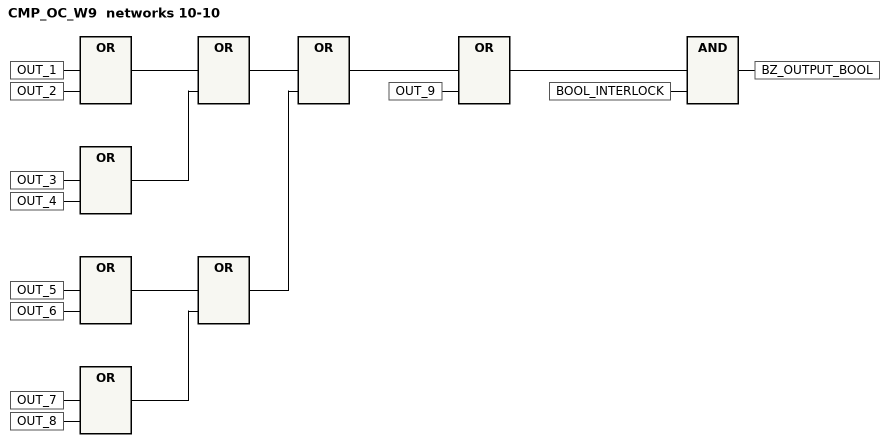
[picture p24: CMP_OC_W9 (FBD) networks 10-10]
_FBD_ (* Function Block Diagram *)
NETWORK 1
	OR(LT(WORD_1, 0), GT(WORD_1, 0)) => OUT_1
NETWORK 2
	OR(LT(WORD_2, 0), GT(WORD_2, 0)) => OUT_2
NETWORK 3
	OR(LT(WORD_3, 0), GT(WORD_3, 0)) => OUT_3
NETWORK 4
	OR(LT(WORD_4, 0), GT(WORD_4, 0)) => OUT_4
NETWORK 5
	OR(LT(WORD_5, 0), GT(WORD_5, 0)) => OUT_5
NETWORK 6
	OR(LT(WORD_6, 0), GT(WORD_6, 0)) => OUT_6
NETWORK 7
	OR(LT(WORD_7, 0), GT(WORD_7, 0)) => OUT_7
NETWORK 8
	OR(LT(WORD_8, 0), GT(WORD_8, 0)) => OUT_8
NETWORK 9
	OR(LT(WORD_9, 0), GT(WORD_9, 0)) => OUT_9
NETWORK 10
	AND(OR(OR(OR(OR(OUT_1, OUT_2), OR(OUT_3, OUT_4)), OR(OR(OUT_5, OUT_6), OR(OUT_7, OUT_8))), OUT_9), BOOL_INTERLOCK) => BZ_OUTPUT_BOOL
_END_FBD_
(* the same logic as Structured Text *)
(* Network 1 *)
OUT_1 := (WORD_1 < 0) OR (WORD_1 > 0);
(* Network 2 *)
OUT_2 := (WORD_2 < 0) OR (WORD_2 > 0);
(* Network 3 *)
OUT_3 := (WORD_3 < 0) OR (WORD_3 > 0);
(* Network 4 *)
OUT_4 := (WORD_4 < 0) OR (WORD_4 > 0);
(* Network 5 *)
OUT_5 := (WORD_5 < 0) OR (WORD_5 > 0);
(* Network 6 *)
OUT_6 := (WORD_6 < 0) OR (WORD_6 > 0);
(* Network 7 *)
OUT_7 := (WORD_7 < 0) OR (WORD_7 > 0);
(* Network 8 *)
OUT_8 := (WORD_8 < 0) OR (WORD_8 > 0);
(* Network 9 *)
OUT_9 := (WORD_9 < 0) OR (WORD_9 > 0);
(* Network 10 *)
BZ_OUTPUT_BOOL := ((((OUT_1 OR OUT_2) OR (OUT_3 OR OUT_4)) OR ((OUT_5 OR OUT_6) OR (OUT_7 OR OUT_8))) OR OUT_9) AND BOOL_INTERLOCK;
END_FUNCTION_BLOCK

(* POU DOWN_COUNT_TIMER, LD *)
FUNCTIONBLOCK DOWN_COUNT_TIMER
VAR_INPUT
	BOOL_SIGNAL_IN: BOOL;
	BOOL_TIMER_RST: BOOL;
	INT_AUTO_RST: INT;
	INT_SV_SEC: INT;
END_VAR
VAR_OUTPUT
	SIGNAL_BOOL: BOOL;
	PV_SEC_INT: INT;
END_VAR
VAR
	DF_1: R_TRIG;
	DF_2: R_TRIG;
	M1: BOOL;
	M2: BOOL;

	T100: TON;
	T101: TON;
	M100: BOOL;
	M101: BOOL;
	M200: BOOL;

	M110: BOOL;
	M300: BOOL;
END_VAR
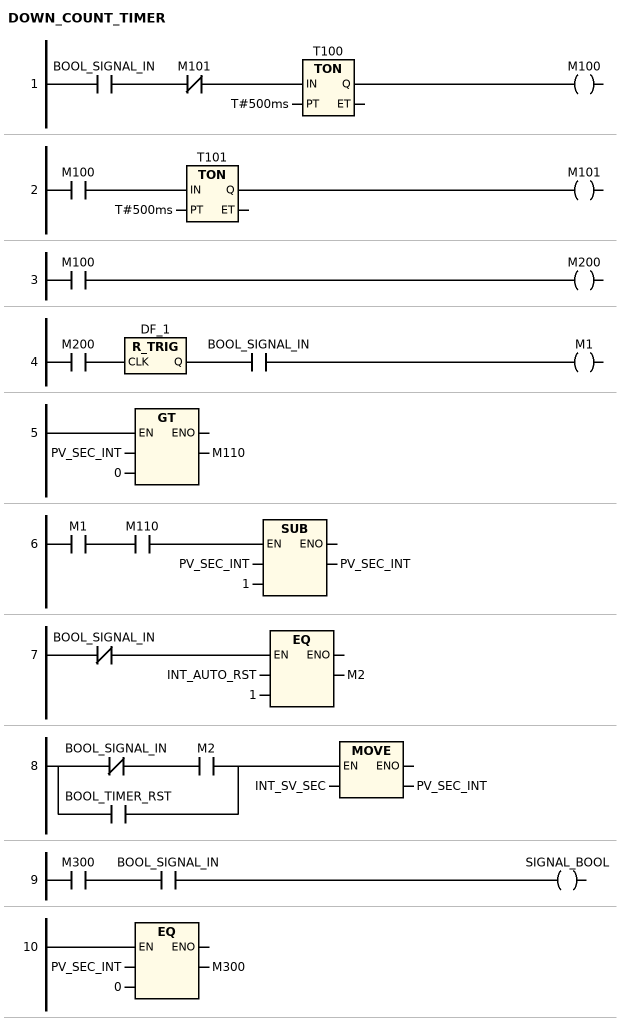
_LD_ (* Ladder Diagram *)
NETWORK 1
	[BOOL_SIGNAL_IN] - [/M101] - T100:TON(IN: *, PT: T#500ms) --- (M100)
NETWORK 2
	[M100] - T101:TON(IN: *, PT: T#500ms) --- (M101)
NETWORK 3
	[M100] --- (M200)
NETWORK 4
	[M200] - DF_1:R_TRIG(CLK: *) - [BOOL_SIGNAL_IN] --- (M1)
NETWORK 5
	*
		EN --- GT(PV_SEC_INT, 0) => M110
NETWORK 6
	[M1] - [M110]
		EN --- SUB(PV_SEC_INT, 1) => PV_SEC_INT
NETWORK 7
	[/BOOL_SIGNAL_IN]
		EN --- EQ(INT_AUTO_RST, 1) => M2
NETWORK 8
	{ [/BOOL_SIGNAL_IN] - [M2] | [BOOL_TIMER_RST] }
		EN --- MOVE(INT_SV_SEC) => PV_SEC_INT
NETWORK 9
	[M300] - [BOOL_SIGNAL_IN] --- (SIGNAL_BOOL)
NETWORK 10
	*
		EN --- EQ(PV_SEC_INT, 0) => M300
_END_LD_
(* the same logic as Structured Text *)
(* Network 1 *)
T100(IN := BOOL_SIGNAL_IN AND NOT M101, PT := T#500ms);
M100 := T100.Q;
(* Network 2 *)
T101(IN := M100, PT := T#500ms);
M101 := T101.Q;
(* Network 3 *)
M200 := M100;
(* Network 4 *)
DF_1(CLK := M200);
M1 := DF_1.Q AND BOOL_SIGNAL_IN;
(* Network 5 *)
M110 := PV_SEC_INT > 0;
(* Network 6 *)
IF M1 AND M110 THEN
	PV_SEC_INT := PV_SEC_INT - 1;
END_IF;
(* Network 7 *)
IF NOT BOOL_SIGNAL_IN THEN
	M2 := INT_AUTO_RST = 1;
END_IF;
(* Network 8 *)
IF NOT BOOL_SIGNAL_IN AND M2 OR BOOL_TIMER_RST THEN
	PV_SEC_INT := INT_SV_SEC;
END_IF;
(* Network 9 *)
SIGNAL_BOOL := M300 AND BOOL_SIGNAL_IN;
(* Network 10 *)
M300 := PV_SEC_INT = 0;
END_FUNCTION_BLOCK

(* POU CLOCK_PLS, LD *)
FUNCTION_BLOCK CLOCK_PLS
VAR_INPUT
	INT_TIME_ms : INT;

END_VAR
VAR_OUTPUT
	CLOCK_PLS_BOOL: BOOL;
END_VAR
VAR
	T0: TON;
	T1: TON;
	M0: BOOL;
	M1: BOOL;
	D0: TIME;
	D1: TIME;
END_VAR
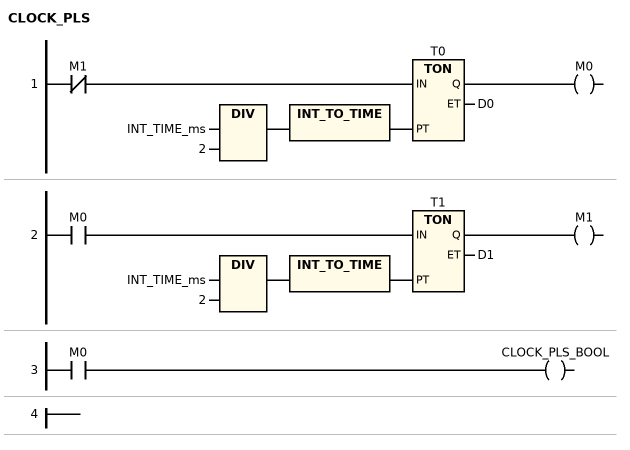
_LD_ (* Ladder Diagram *)
NETWORK 1
	[/M1] - T0:TON(IN: *, PT: INT_TO_TIME(DIV(INT_TIME_ms, 2)), ET => D0) --- (M0)
NETWORK 2
	[M0] - T1:TON(IN: *, PT: INT_TO_TIME(DIV(INT_TIME_ms, 2)), ET => D1) --- (M1)
NETWORK 3
	[M0] --- (CLOCK_PLS_BOOL)
NETWORK 4
	*
_END_LD_
(* the same logic as Structured Text *)
(* Network 1 *)
T0(IN := NOT M1, PT := INT_TO_TIME(INT_TIME_ms / 2));
D0 := T0.ET;
M0 := T0.Q;
(* Network 2 *)
T1(IN := M0, PT := INT_TO_TIME(INT_TIME_ms / 2));
D1 := T1.ET;
M1 := T1.Q;
(* Network 3 *)
CLOCK_PLS_BOOL := M0;
(* Network 4 *)
END_FUNCTION_BLOCK

(* POU DC_PID_FB, LD *)
FUNCTION_BLOCK DC_PID_FB
VAR_INPUT
	BOOL_LOW_FLOW_EN : BOOL;
	INT_HIGH_FLOW_LPM : INT;
	INT_LOW_FLOW_LPM : INT;
	INT_H_L_FLOW_RATIO : INT;
	INT_D1_LPM : INT;
	INT_D2_LPM : INT;
	INT_D3_LPM : INT;
	INT_D4_RAW : INT;
	INT_D5_RAW : INT;
	INT_D6_RAW : INT;
	INT_D1_RATIO : INT;
	INT_D2_RATIO : INT;
	INT_D3_RATIO : INT;
	INT_D4_RATIO : INT;
	INT_D5_RATIO : INT;
	INT_D6_RATIO : INT;

END_VAR

VAR_OUTPUT

	PID_FLOW_RAW : INT;
	D1_RAW_INT : INT;
	D2_RAW_INT : INT;
	D3_RAW_INT : INT;
	D4_LPM_INT : INT;
	D5_LPM_INT : INT;
	D6_LPM_INT : INT;

END_VAR
VAR
	D5EN: BOOL;
	D4EN: BOOL;
	D6EN: BOOL;
	D4REN: BOOL;
	D5REN: BOOL;
	D6REN: BOOL;
END_VAR
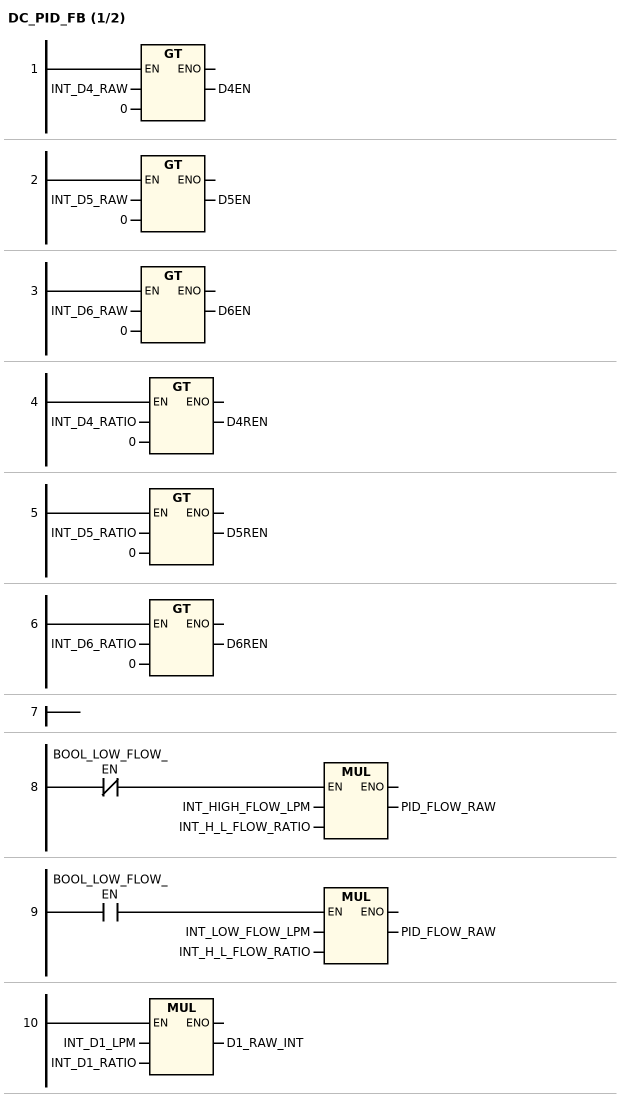
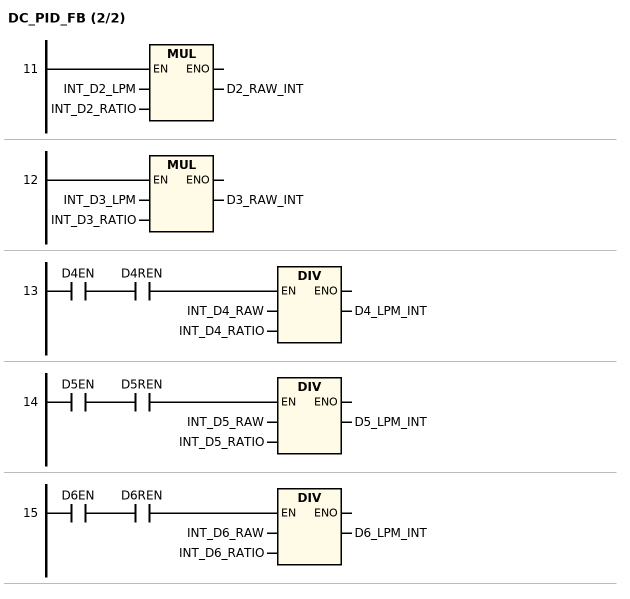
_LD_ (* Ladder Diagram *)
NETWORK 1
	*
		EN --- GT(INT_D4_RAW, 0) => D4EN
NETWORK 2
	*
		EN --- GT(INT_D5_RAW, 0) => D5EN
NETWORK 3
	*
		EN --- GT(INT_D6_RAW, 0) => D6EN
NETWORK 4
	*
		EN --- GT(INT_D4_RATIO, 0) => D4REN
NETWORK 5
	*
		EN --- GT(INT_D5_RATIO, 0) => D5REN
NETWORK 6
	*
		EN --- GT(INT_D6_RATIO, 0) => D6REN
NETWORK 7
	*
NETWORK 8
	[/BOOL_LOW_FLOW_EN]
		EN --- MUL(INT_HIGH_FLOW_LPM, INT_H_L_FLOW_RATIO) => PID_FLOW_RAW
NETWORK 9
	[BOOL_LOW_FLOW_EN]
		EN --- MUL(INT_LOW_FLOW_LPM, INT_H_L_FLOW_RATIO) => PID_FLOW_RAW
NETWORK 10
	*
		EN --- MUL(INT_D1_LPM, INT_D1_RATIO) => D1_RAW_INT
NETWORK 11
	*
		EN --- MUL(INT_D2_LPM, INT_D2_RATIO) => D2_RAW_INT
NETWORK 12
	*
		EN --- MUL(INT_D3_LPM, INT_D3_RATIO) => D3_RAW_INT
NETWORK 13
	[D4EN] - [D4REN]
		EN --- DIV(INT_D4_RAW, INT_D4_RATIO) => D4_LPM_INT
NETWORK 14
	[D5EN] - [D5REN]
		EN --- DIV(INT_D5_RAW, INT_D5_RATIO) => D5_LPM_INT
NETWORK 15
	[D6EN] - [D6REN]
		EN --- DIV(INT_D6_RAW, INT_D6_RATIO) => D6_LPM_INT
_END_LD_
(* the same logic as Structured Text *)
(* Network 1 *)
D4EN := INT_D4_RAW > 0;
(* Network 2 *)
D5EN := INT_D5_RAW > 0;
(* Network 3 *)
D6EN := INT_D6_RAW > 0;
(* Network 4 *)
D4REN := INT_D4_RATIO > 0;
(* Network 5 *)
D5REN := INT_D5_RATIO > 0;
(* Network 6 *)
D6REN := INT_D6_RATIO > 0;
(* Network 7 *)
(* Network 8 *)
IF NOT BOOL_LOW_FLOW_EN THEN
	PID_FLOW_RAW := INT_HIGH_FLOW_LPM * INT_H_L_FLOW_RATIO;
END_IF;
(* Network 9 *)
IF BOOL_LOW_FLOW_EN THEN
	PID_FLOW_RAW := INT_LOW_FLOW_LPM * INT_H_L_FLOW_RATIO;
END_IF;
(* Network 10 *)
D1_RAW_INT := INT_D1_LPM * INT_D1_RATIO;
(* Network 11 *)
D2_RAW_INT := INT_D2_LPM * INT_D2_RATIO;
(* Network 12 *)
D3_RAW_INT := INT_D3_LPM * INT_D3_RATIO;
(* Network 13 *)
IF D4EN AND D4REN THEN
	D4_LPM_INT := INT_D4_RAW / INT_D4_RATIO;
END_IF;
(* Network 14 *)
IF D5EN AND D5REN THEN
	D5_LPM_INT := INT_D5_RAW / INT_D5_RATIO;
END_IF;
(* Network 15 *)
IF D6EN AND D6REN THEN
	D6_LPM_INT := INT_D6_RAW / INT_D6_RATIO;
END_IF;
END_FUNCTION_BLOCK

(* POU EQ_GT, LD *)
FUNCTION_BLOCK EQ_GT
VAR_INPUT
	INT_SOURCE_A: INT;
	INT_SOURCE_B: INT;
END_VAR
VAR_OUTPUT
	SIGNAL_BOOL: BOOL;
END_VAR
VAR
	M0: BOOL;
	M1: BOOL;
END_VAR
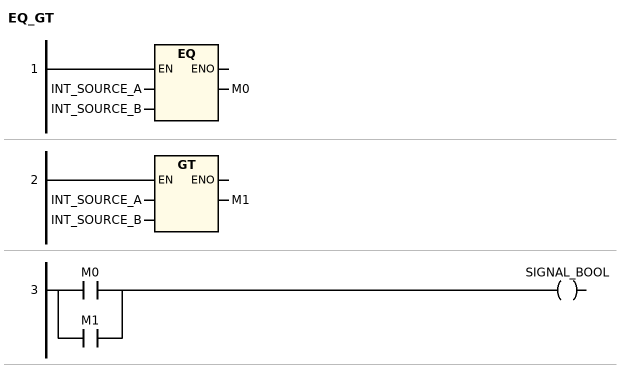
_LD_ (* Ladder Diagram *)
NETWORK 1
	*
		EN --- EQ(INT_SOURCE_A, INT_SOURCE_B) => M0
NETWORK 2
	*
		EN --- GT(INT_SOURCE_A, INT_SOURCE_B) => M1
NETWORK 3
	{ [M0] | [M1] } --- (SIGNAL_BOOL)
_END_LD_
(* the same logic as Structured Text *)
(* Network 1 *)
M0 := INT_SOURCE_A = INT_SOURCE_B;
(* Network 2 *)
M1 := INT_SOURCE_A > INT_SOURCE_B;
(* Network 3 *)
SIGNAL_BOOL := M0 OR M1;
END_FUNCTION_BLOCK

(* POU EQ_LT, LD *)
FUNCTION_BLOCK EQ_LT
VAR_INPUT
	INT_SOURCE_A:INT;
	INT_SOURCE_B:INT;
END_VAR
VAR_OUTPUT
	SIGNAL_BOOL:BOOL;
END_VAR
VAR
	M0: BOOL;
	M1: BOOL;
END_VAR
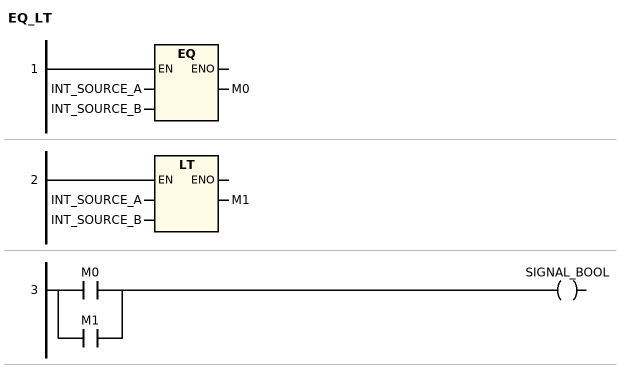
_LD_ (* Ladder Diagram *)
NETWORK 1
	*
		EN --- EQ(INT_SOURCE_A, INT_SOURCE_B) => M0
NETWORK 2
	*
		EN --- LT(INT_SOURCE_A, INT_SOURCE_B) => M1
NETWORK 3
	{ [M0] | [M1] } --- (SIGNAL_BOOL)
_END_LD_
(* the same logic as Structured Text *)
(* Network 1 *)
M0 := INT_SOURCE_A = INT_SOURCE_B;
(* Network 2 *)
M1 := INT_SOURCE_A < INT_SOURCE_B;
(* Network 3 *)
SIGNAL_BOOL := M0 OR M1;
END_FUNCTION_BLOCK

(* POU INDIRECT_FN, LD *)
FUNCTION_BLOCK INDIRECT_FN
VAR_INPUT
	BOOL_SV_PB: BOOL;		(*SAVE PB (TS)*)
	BOOL_LD_PB: BOOL;			(*LOAD PB (TS)*)
	INT_P_NO: INT;		(*PROGRAM NO (TS) 1~10*)
	INT_D00:INT;
	INT_D01:INT;
	INT_D02:INT;
	INT_D03:INT;
	INT_D04:INT;
	INT_D05:INT;
	INT_D06:INT;
	INT_D07:INT;
	INT_D08:INT;
	INT_D09:INT;
	INT_D10:INT;
	INT_D11:INT;
	INT_D12:INT;
	INT_D13:INT;
	INT_D14:INT;
	INT_D15:INT;
	INT_D16:INT;
	INT_D17:INT;
	INT_D18:INT;
	INT_D19:INT;
	INT_D20:INT;
	INT_D21:INT;
	INT_D22:INT;
	INT_D23:INT;
	INT_D24:INT;
	INT_D25:INT;
	INT_D26:INT;
	INT_D27:INT;
	INT_D28:INT;
	INT_D29:INT;
	INT_D30:INT;
	STG_STG1:STRING;
END_VAR
VAR_OUTPUT
	SV_PB_IND_BOOL:BOOL;
	LD_PB_IND_BOOL:BOOL;
	D00_INT:INT;
	D01_INT:INT;
	D02_INT:INT;
	D03_INT:INT;
	D04_INT:INT;
	D05_INT:INT;
	D06_INT:INT;
	D07_INT:INT;
	D08_INT:INT;
	D09_INT:INT;
	D10_INT:INT;
	D11_INT:INT;
	D12_INT:INT;
	D13_INT:INT;
	D14_INT:INT;
	D15_INT:INT;
	D16_INT:INT;
	D17_INT:INT;
	D18_INT:INT;
	D19_INT:INT;
	D20_INT:INT;
	D21_INT:INT;
	D22_INT:INT;
	D23_INT:INT;
	D24_INT:INT;
	D25_INT:INT;
	D26_INT:INT;
	D27_INT:INT;
	D28_INT:INT;
	D29_INT:INT;
	D30_INT:INT;
	STG1_STG:STRING;
END_VAR
VAR

	P1B: BOOL;
	P2B: BOOL;
	P3B: BOOL;
	P4B: BOOL;
	P5B: BOOL;
	P6B: BOOL;
	P7B: BOOL;
	P8B: BOOL;
	P9B: BOOL;
	P10B: BOOL;
	SV_HR: BOOL;
	SV_T: TON;
	SV_CR: BOOL;
	LD_HR: BOOL;
	LD_CR: BOOL;
	LD_T: TON;
	SV_DF: R_TRIG;
	SV_PLS: BOOL;
	LD_DF: R_TRIG;
	LD_PLS: BOOL;
	ALWAYS_ON: BOOL;
	TPC: TON;
	N0: BOOL;
	TPC1: TON;
	N1: BOOL;
	CNG_P_NO: INT;
	NPC: BOOL;		(*NON PROGRAM CHANGE*)
	PCDF: R_TRIG;
	PCTDF: BOOL;
	PCDFN: F_TRIG;
	PC_PLS: BOOL;
	SVPLS: R_TRIG;
	SV_PB_PLS: BOOL;
	LDPLS: R_TRIG;
	LD_PB_PLS: BOOL;
END_VAR
VAR RETAIN
	P01D00:INT;
	P01D01:INT;
	P01D02:INT;
	P01D03:INT;
	P01D04:INT;
	P01D05:INT;
	P01D06:INT;
	P01D07:INT;
	P01D08:INT;
	P01D09:INT;
	P01D10:INT;
	P01D11:INT;
	P01D12:INT;
	P01D13:INT;
	P01D14:INT;
	P01D15:INT;
	P01D16:INT;
	P01D17:INT;
	P01D18:INT;
	P01D19:INT;
	P01D20:INT;
	P01D21:INT;
	P01D22:INT;
	P01D23:INT;
	P01D24:INT;
	P01D25:INT;
	P01D26:INT;
	P01D27:INT;
	P01D28:INT;
	P01D29:INT;
	P01D30:INT;
	P01STG:STRING;
	P02D00:INT;
	P02D01:INT;
	P02D02:INT;
	P02D03:INT;
	P02D04:INT;
	P02D05:INT;
	P02D06:INT;
	P02D07:INT;
	P02D08:INT;
	P02D09:INT;
	P02D10:INT;
	P02D11:INT;
	P02D12:INT;
	P02D13:INT;
	P02D14:INT;
	P02D15:INT;
	P02D16:INT;
	P02D17:INT;
	P02D18:INT;
	P02D19:INT;
	P02D20:INT;
	P02D21:INT;
	P02D22:INT;
	P02D23:INT;
	P02D24:INT;
	P02D25:INT;
	P02D26:INT;
	P02D27:INT;
	P02D28:INT;
	P02D29:INT;
	P02D30:INT;
	P02STG:STRING;
	P03D00:INT;
	P03D01:INT;
	P03D02:INT;
	P03D03:INT;
	P03D04:INT;
	P03D05:INT;
	P03D06:INT;
	P03D07:INT;
	P03D08:INT;
	P03D09:INT;
	P03D10:INT;
	P03D11:INT;
	P03D12:INT;
	P03D13:INT;
	P03D14:INT;
	P03D15:INT;
	P03D16:INT;
	P03D17:INT;
	P03D18:INT;
	P03D19:INT;
	P03D20:INT;
	P03D21:INT;
	P03D22:INT;
	P03D23:INT;
	P03D24:INT;
	P03D25:INT;
	P03D26:INT;
	P03D27:INT;
	P03D28:INT;
	P03D29:INT;
	P03D30:INT;
	P03STG:STRING;
	P04D00:INT;
	P04D01:INT;
	P04D02:INT;
	P04D03:INT;
	P04D04:INT;
	P04D05:INT;
	P04D06:INT;
	P04D07:INT;
	P04D08:INT;
	P04D09:INT;
	P04D10:INT;
	P04D11:INT;
	P04D12:INT;
	P04D13:INT;
	P04D14:INT;
	P04D15:INT;
	P04D16:INT;
	P04D17:INT;
	P04D18:INT;
	P04D19:INT;
	P04D20:INT;
	P04D21:INT;
	P04D22:INT;
	P04D23:INT;
	P04D24:INT;
	P04D25:INT;
	P04D26:INT;
	P04D27:INT;
	P04D28:INT;
	P04D29:INT;
	P04D30:INT;
	P04STG:STRING;
	P05D00:INT;
	P05D01:INT;
	P05D02:INT;
	P05D03:INT;
	P05D04:INT;
	P05D05:INT;
	P05D06:INT;
	P05D07:INT;
	P05D08:INT;
	P05D09:INT;
	P05D10:INT;
	P05D11:INT;
	P05D12:INT;
	P05D13:INT;
	P05D14:INT;
	P05D15:INT;
	P05D16:INT;
	P05D17:INT;
	P05D18:INT;
	P05D19:INT;
	P05D20:INT;
	P05D21:INT;
	P05D22:INT;
	P05D23:INT;
	P05D24:INT;
	P05D25:INT;
	P05D26:INT;
	P05D27:INT;
	P05D28:INT;
	P05D29:INT;
	P05D30:INT;
	P05STG:STRING;
	P06D00:INT;
	P06D01:INT;
	P06D02:INT;
	P06D03:INT;
	P06D04:INT;
	P06D05:INT;
	P06D06:INT;
	P06D07:INT;
	P06D08:INT;
	P06D09:INT;
	P06D10:INT;
	P06D11:INT;
	P06D12:INT;
	P06D13:INT;
	P06D14:INT;
	P06D15:INT;
	P06D16:INT;
	P06D17:INT;
	P06D18:INT;
	P06D19:INT;
	P06D20:INT;
	P06D21:INT;
	P06D22:INT;
	P06D23:INT;
	P06D24:INT;
	P06D25:INT;
	P06D26:INT;
	P06D27:INT;
	P06D28:INT;
	P06D29:INT;
	P06D30:INT;
	P06STG:STRING;
	P07D00:INT;
	P07D01:INT;
	P07D02:INT;
	P07D03:INT;
	P07D04:INT;
	P07D05:INT;
	P07D06:INT;
	P07D07:INT;
	P07D08:INT;
	P07D09:INT;
	P07D10:INT;
	P07D11:INT;
	P07D12:INT;
	P07D13:INT;
	P07D14:INT;
	P07D15:INT;
	P07D16:INT;
	P07D17:INT;
	P07D18:INT;
	P07D19:INT;
	P07D20:INT;
	P07D21:INT;
	P07D22:INT;
	P07D23:INT;
	P07D24:INT;
	P07D25:INT;
	P07D26:INT;
	P07D27:INT;
	P07D28:INT;
	P07D29:INT;
	P07D30:INT;
	P07STG:STRING;
	P08D00:INT;
	P08D01:INT;
	P08D02:INT;
	P08D03:INT;
	P08D04:INT;
	P08D05:INT;
	P08D06:INT;
	P08D07:INT;
	P08D08:INT;
	P08D09:INT;
	P08D10:INT;
	P08D11:INT;
	P08D12:INT;
	P08D13:INT;
	P08D14:INT;
	P08D15:INT;
	P08D16:INT;
	P08D17:INT;
	P08D18:INT;
	P08D19:INT;
	P08D20:INT;
	P08D21:INT;
	P08D22:INT;
	P08D23:INT;
	P08D24:INT;
	P08D25:INT;
	P08D26:INT;
	P08D27:INT;
	P08D28:INT;
	P08D29:INT;
	P08D30:INT;
	P08STG:STRING;
	P09D00:INT;
	P09D01:INT;
	P09D02:INT;
	P09D03:INT;
	P09D04:INT;
	P09D05:INT;
	P09D06:INT;
	P09D07:INT;
	P09D08:INT;
	P09D09:INT;
	P09D10:INT;
	P09D11:INT;
	P09D12:INT;
	P09D13:INT;
	P09D14:INT;
	P09D15:INT;
	P09D16:INT;
	P09D17:INT;
	P09D18:INT;
	P09D19:INT;
	P09D20:INT;
	P09D21:INT;
	P09D22:INT;
	P09D23:INT;
	P09D24:INT;
	P09D25:INT;
	P09D26:INT;
	P09D27:INT;
	P09D28:INT;
	P09D29:INT;
	P09D30:INT;
	P09STG:STRING;
	P10D00:INT;
	P10D01:INT;
	P10D02:INT;
	P10D03:INT;
	P10D04:INT;
	P10D05:INT;
	P10D06:INT;
	P10D07:INT;
	P10D08:INT;
	P10D09:INT;
	P10D10:INT;
	P10D11:INT;
	P10D12:INT;
	P10D13:INT;
	P10D14:INT;
	P10D15:INT;
	P10D16:INT;
	P10D17:INT;
	P10D18:INT;
	P10D19:INT;
	P10D20:INT;
	P10D21:INT;
	P10D22:INT;
	P10D23:INT;
	P10D24:INT;
	P10D25:INT;
	P10D26:INT;
	P10D27:INT;
	P10D28:INT;
	P10D29:INT;
	P10D30:INT;
	P10STG:STRING;

END_VAR
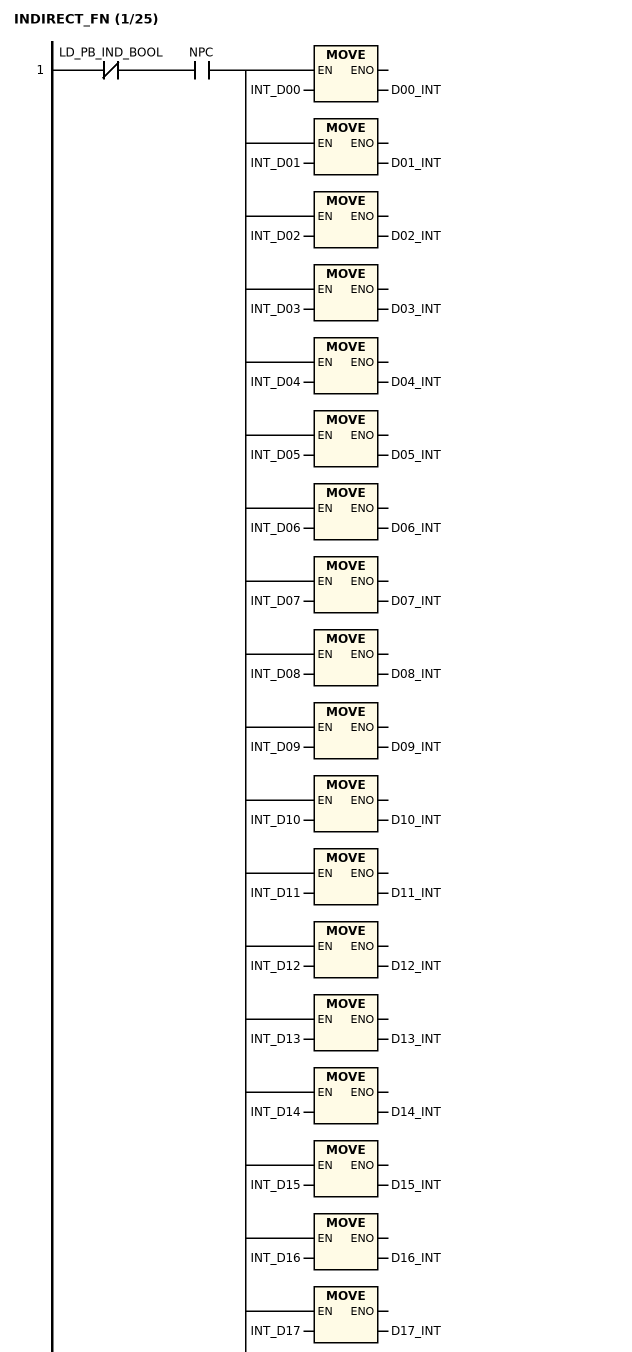
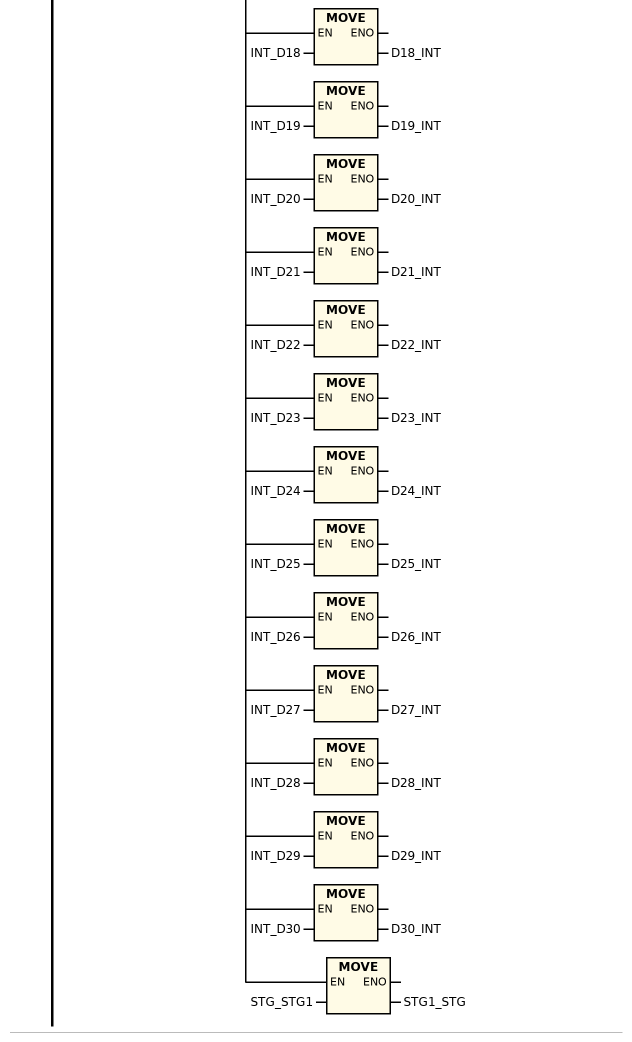
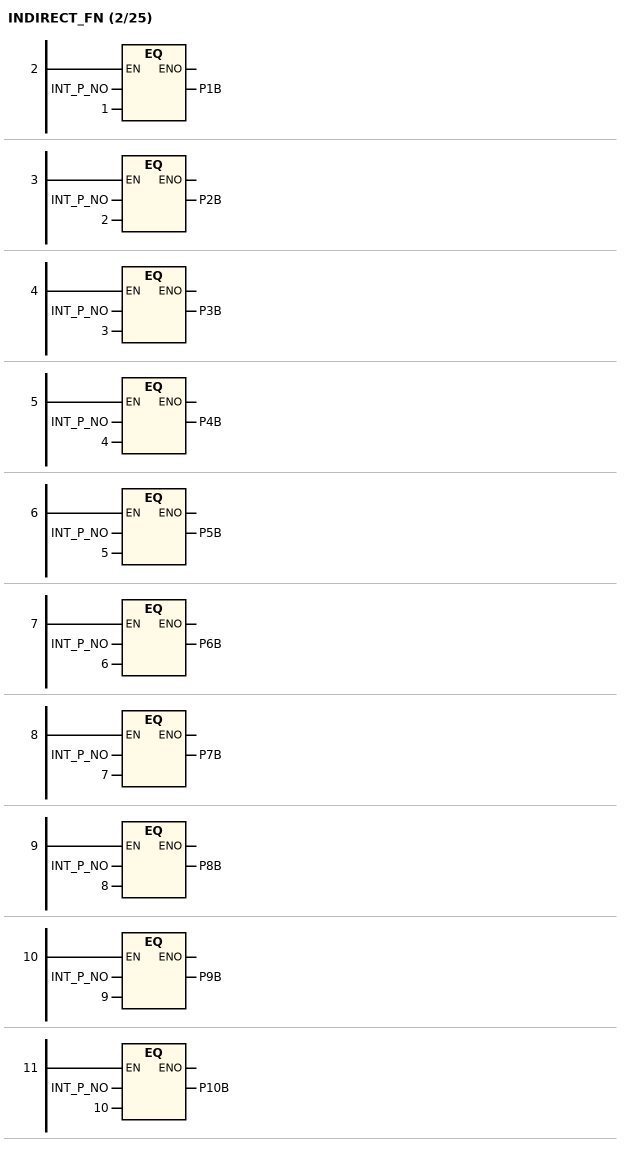
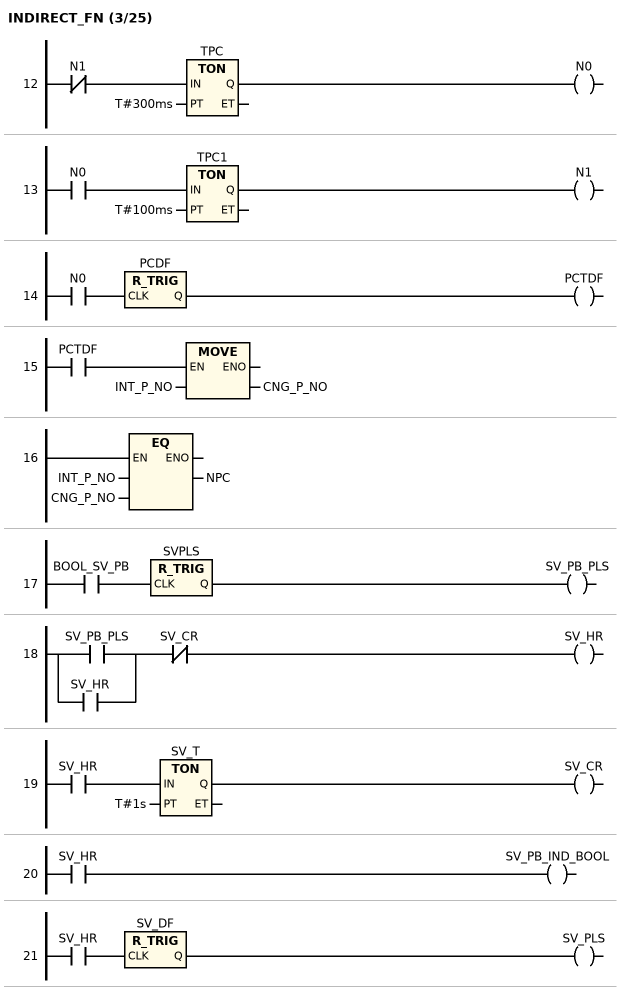
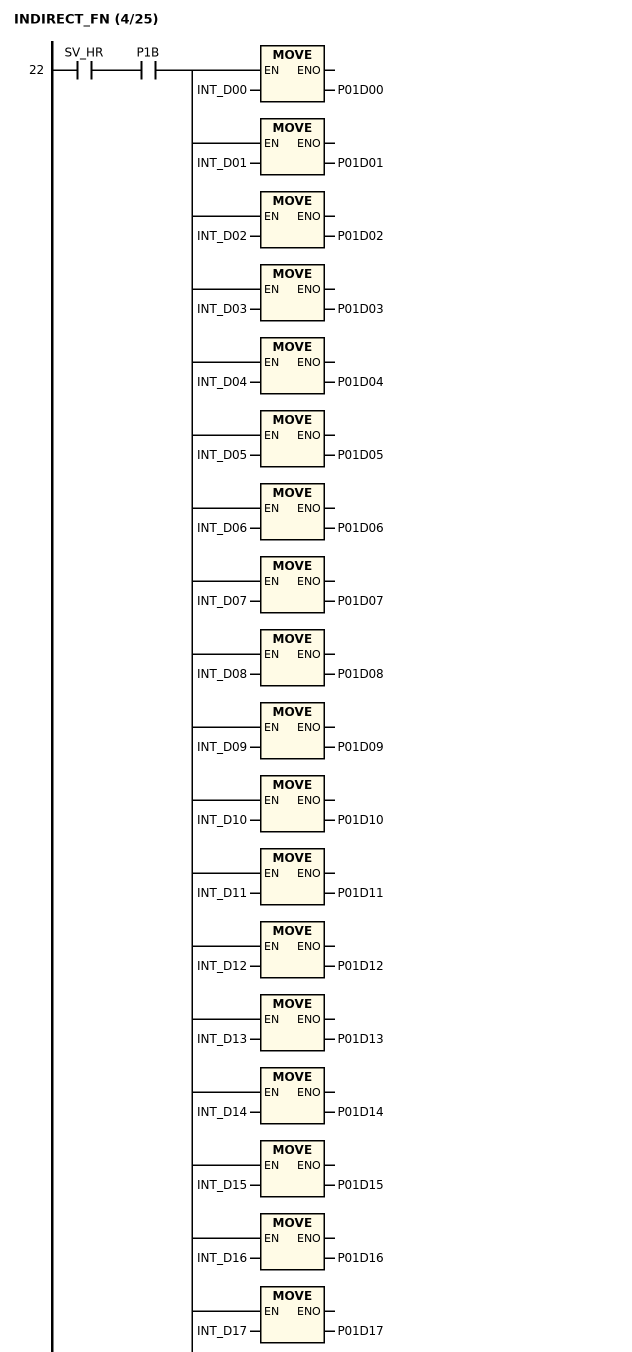
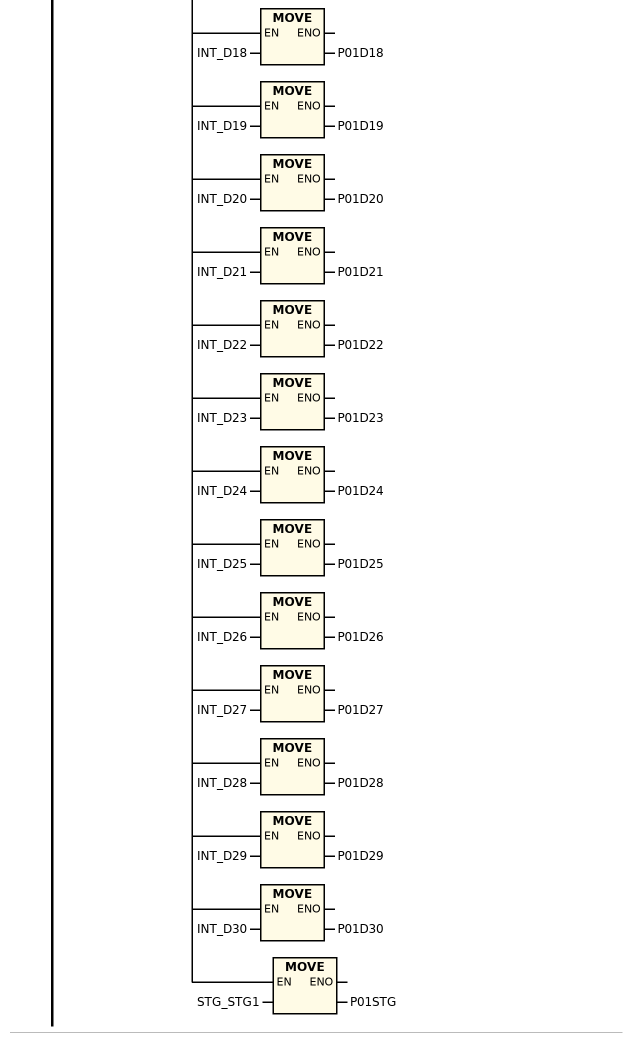
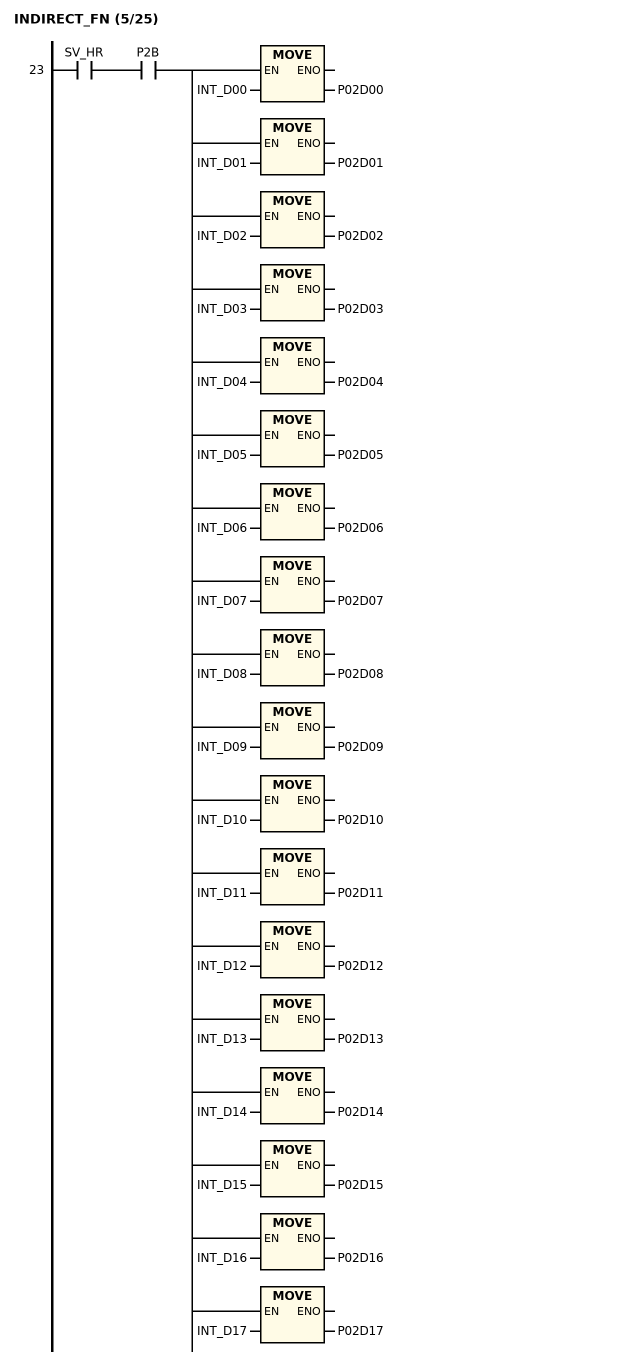
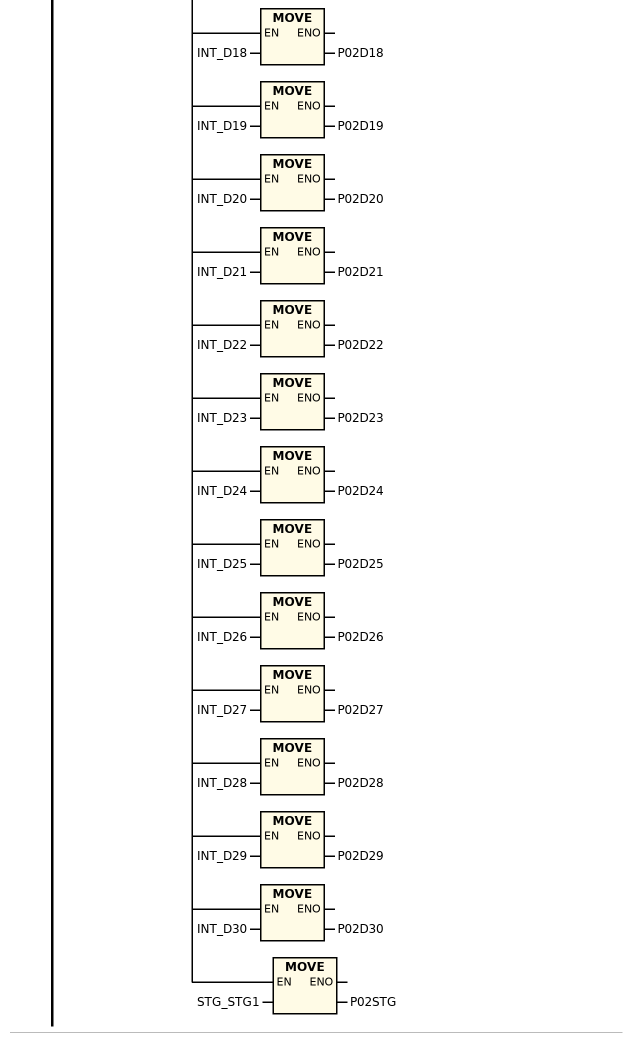
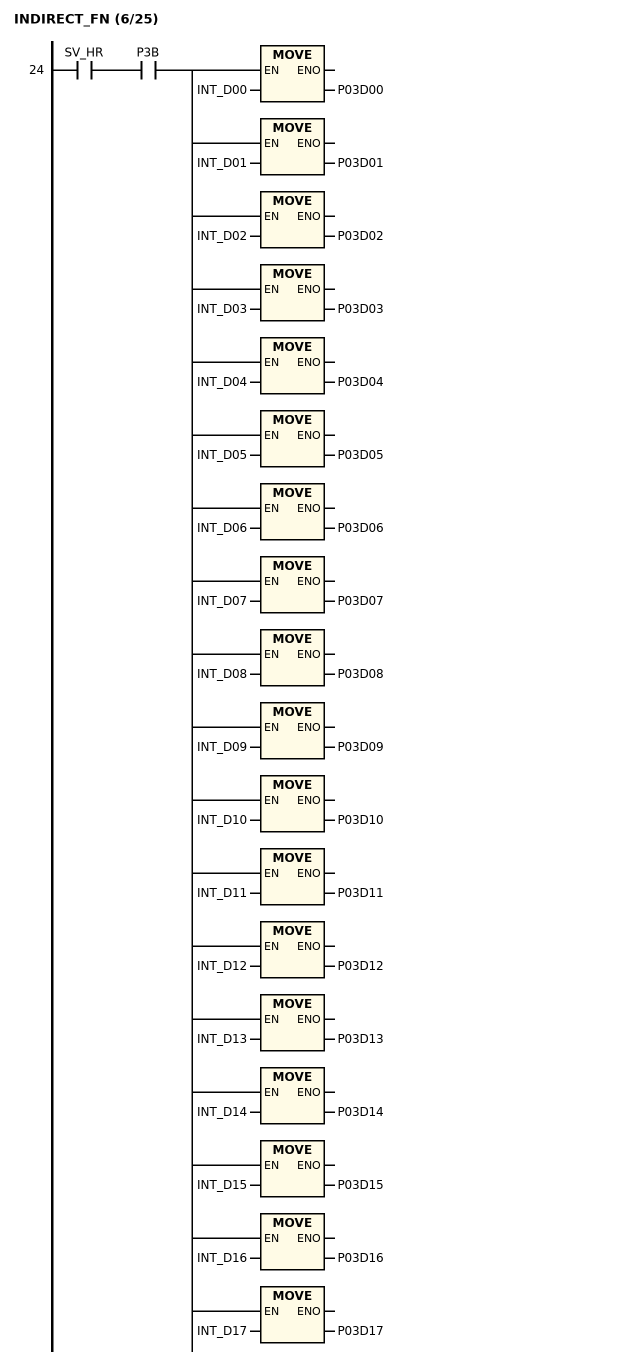
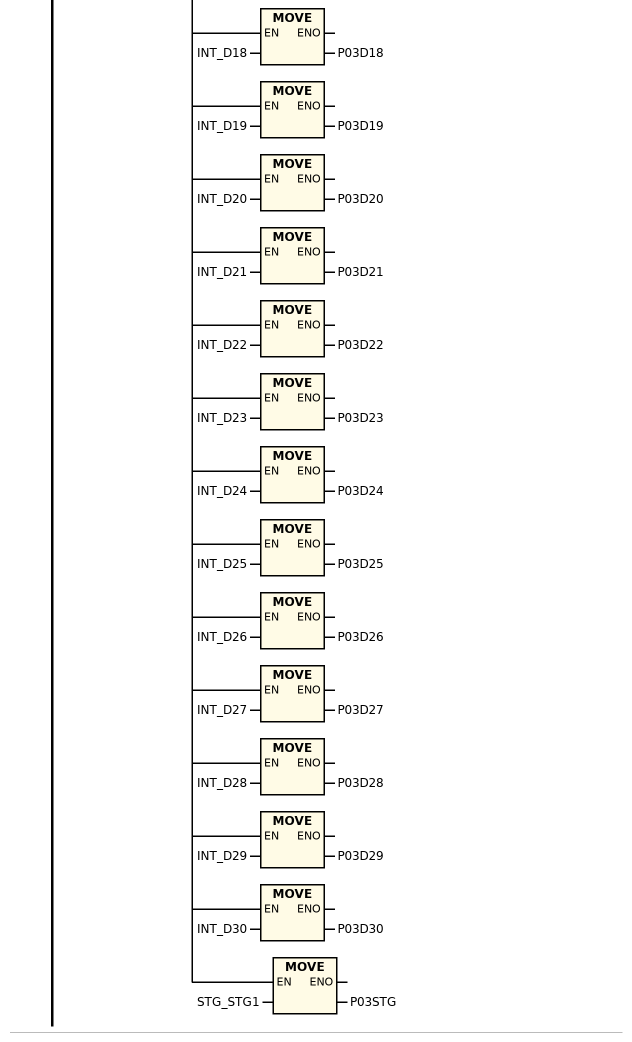
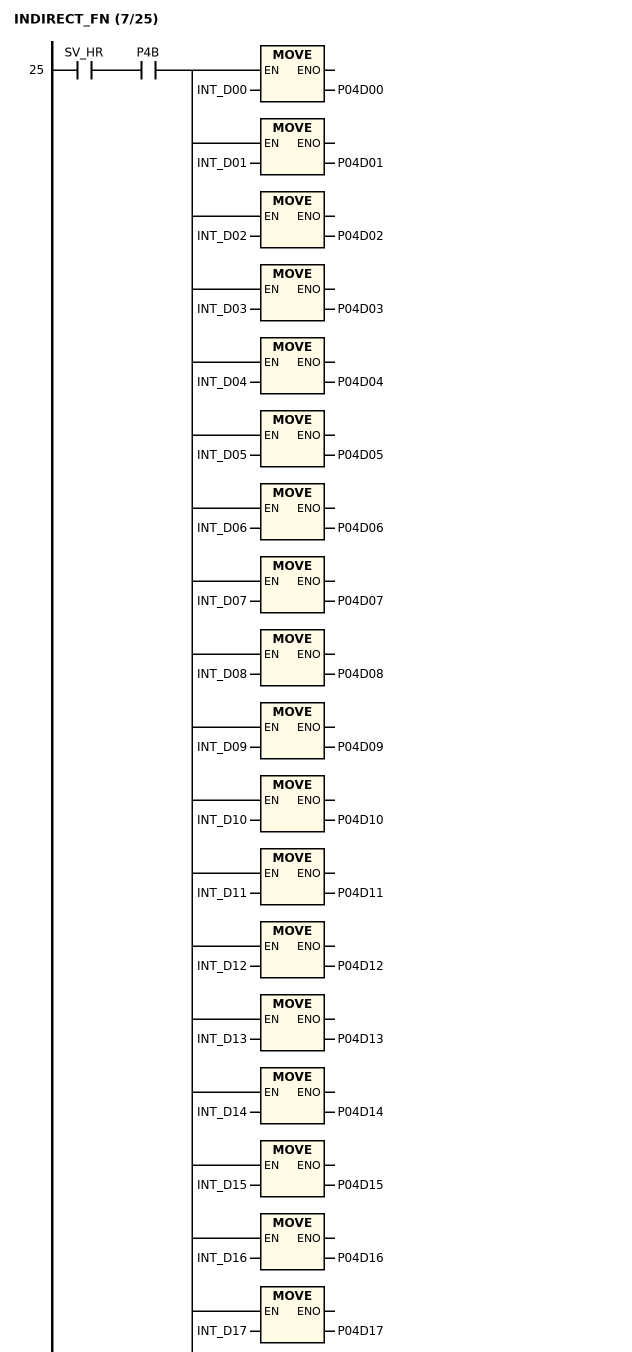
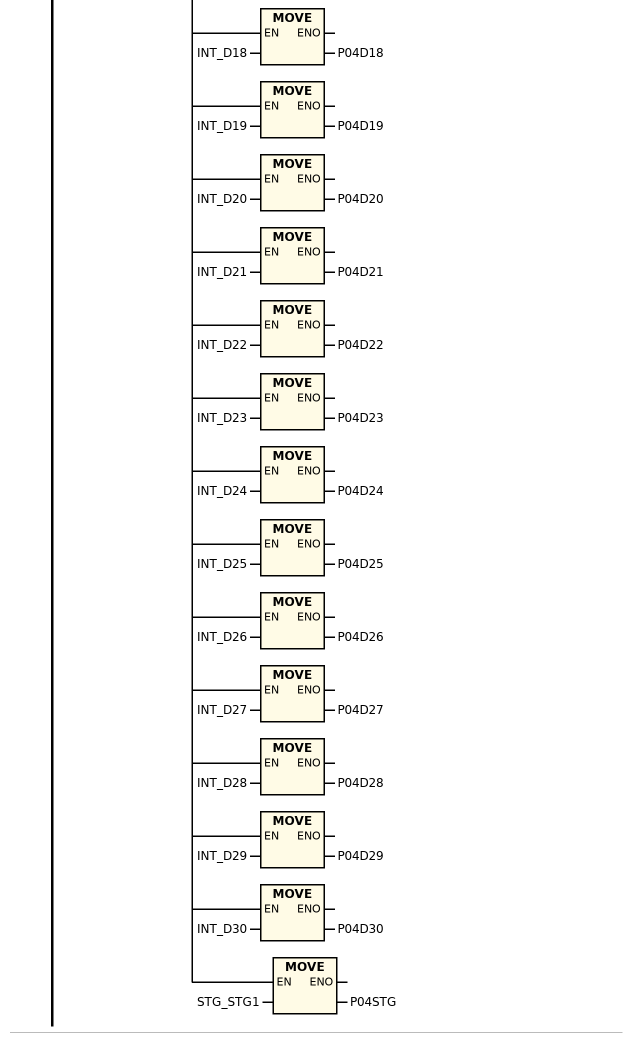
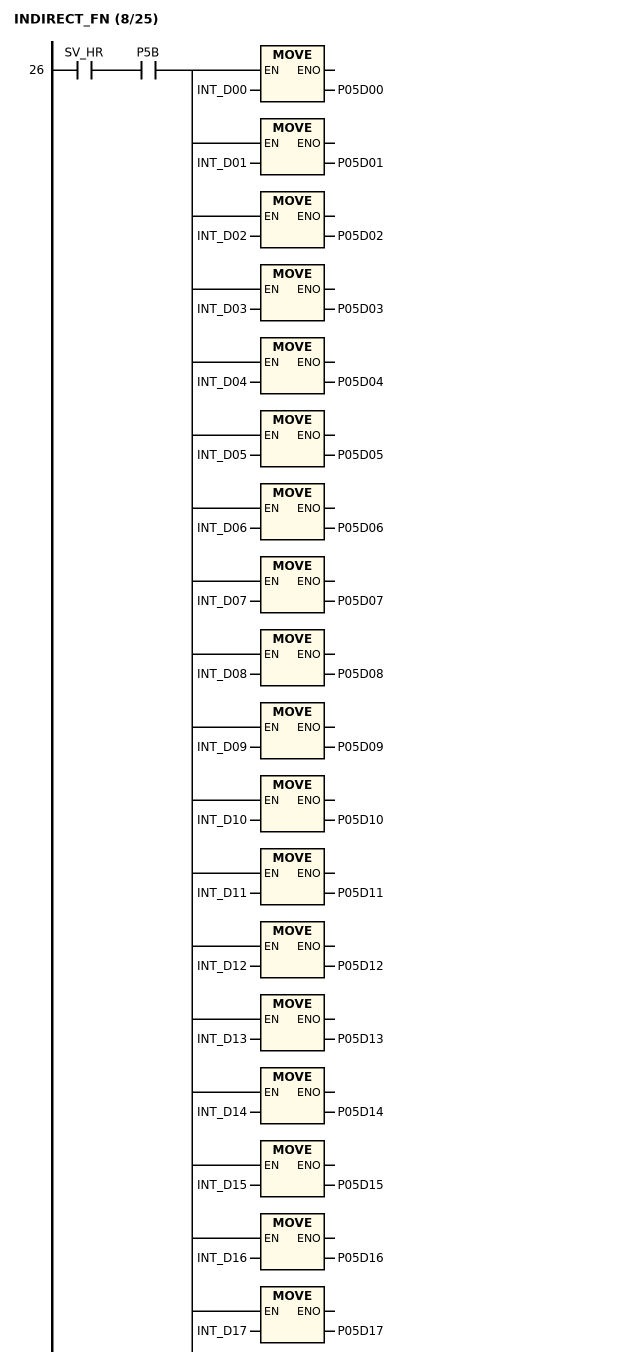
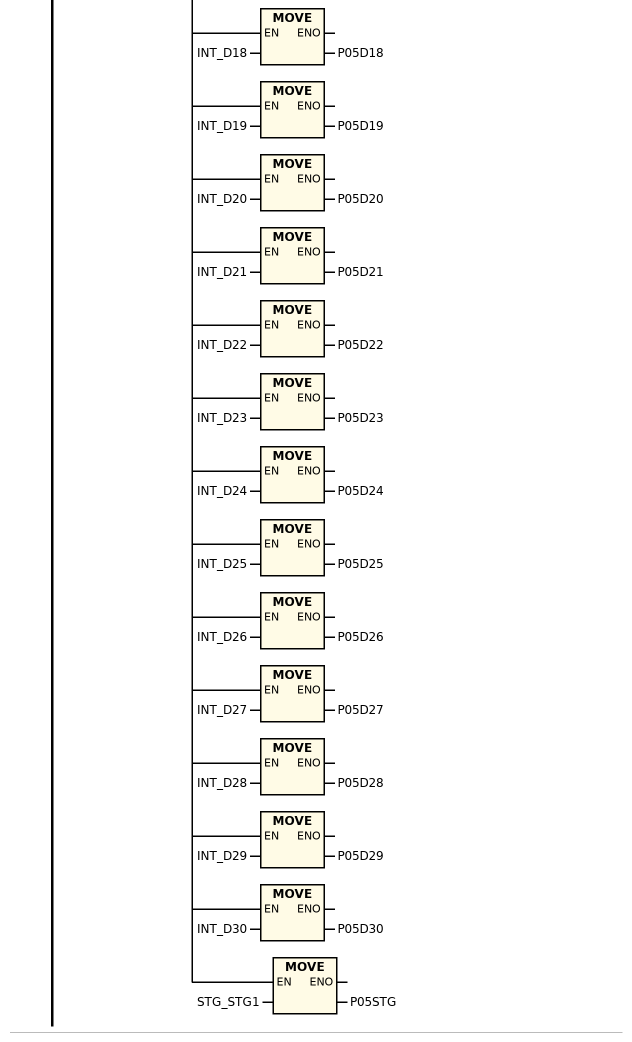
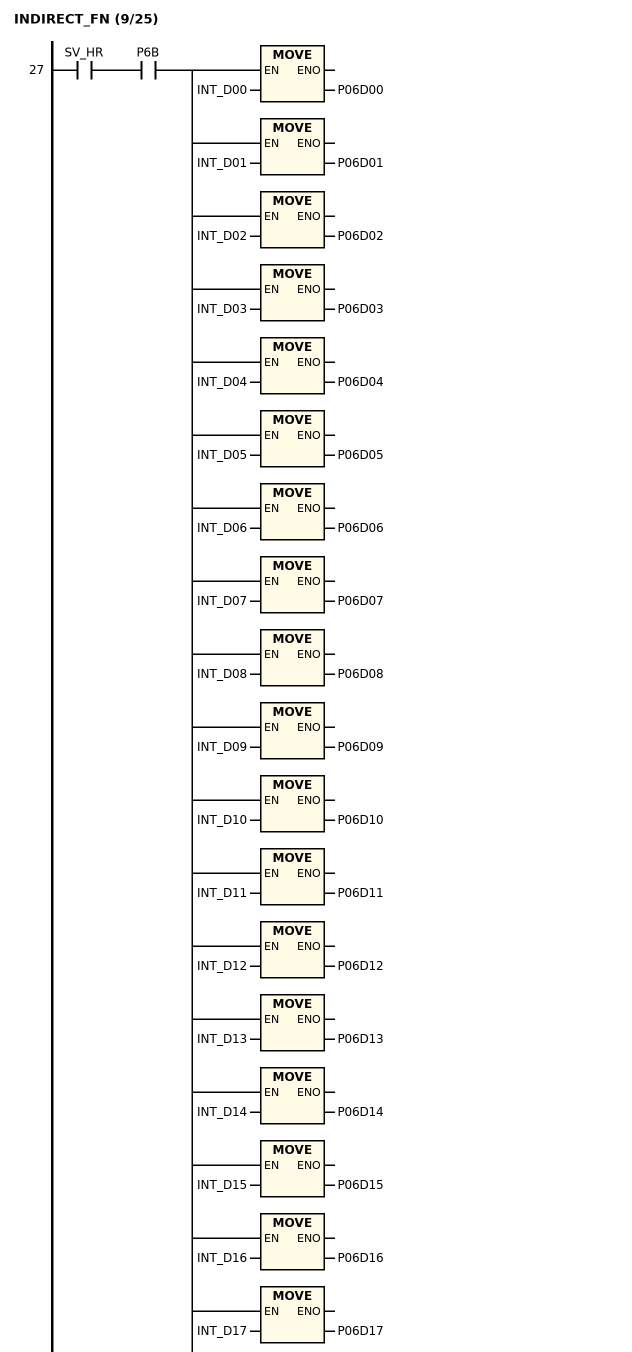
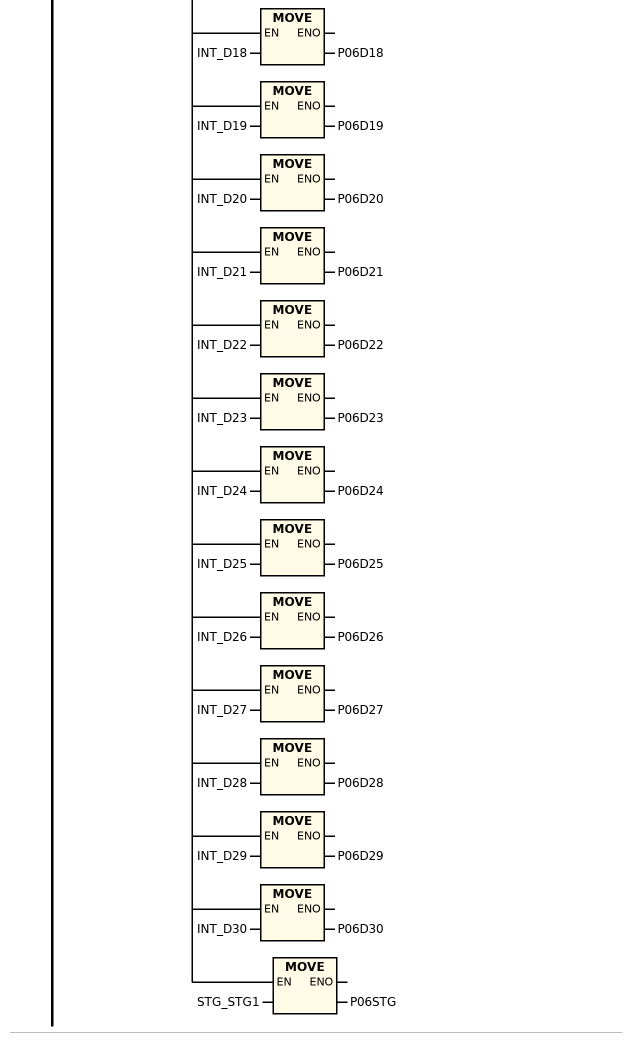
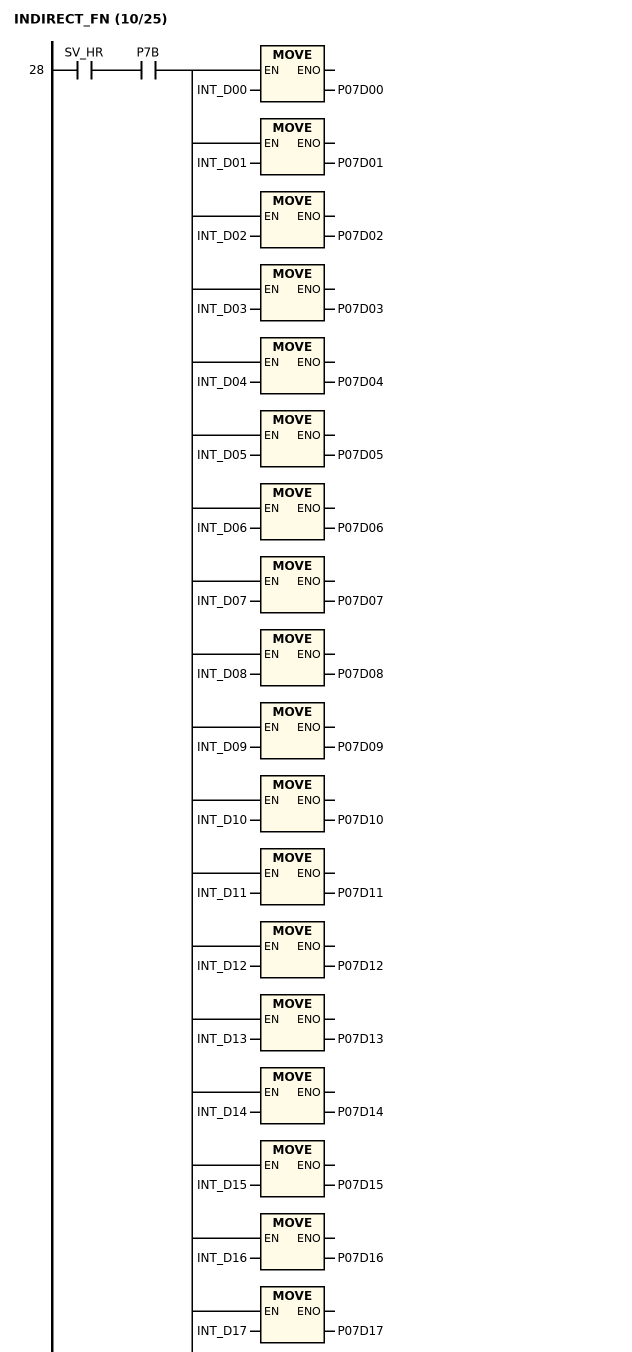
